SUBAPPLICATION Uebung_003e_AX (* DigitalInput_I1-4 auf DigitalOutput_Q1-4 - flach mit Adapter mit Bypass (Druckumlaufventil) *)
  (* Standard: 61499-2; Description: Copyright (c) 2023 Meisterschulen am Ostbahnhof This program and the accompanying materials are made available under the terms of the Eclipse Public License 2.0 which is available at https://www.eclipse.org/legal/epl-2.0/ SPDX-License-Identifier: EPL-2.0 *)
  (* Version 1.0, 2023-10-23, Franz Höpfinger, Meisterschulen am Ostbahnhof, initial API and implementation and/or initial documentation *)
  PACKAGE Uebungen;
  IMPORT logiBUS::io::DI::logiBUS_DI::Input_I1;
  IMPORT logiBUS::io::DI::logiBUS_DI::Input_I2;
  IMPORT logiBUS::io::DI::logiBUS_DI::Input_I3;
  IMPORT logiBUS::io::DI::logiBUS_DI::Input_I4;
  IMPORT logiBUS::io::DQ::logiBUS_DO::Output_Q1;
  IMPORT logiBUS::io::DQ::logiBUS_DO::Output_Q2;
  IMPORT logiBUS::io::DQ::logiBUS_DO::Output_Q3;
  IMPORT logiBUS::io::DQ::logiBUS_DO::Output_Q4;
  IMPORT logiBUS::io::DQ::logiBUS_DO::Output_Q8;
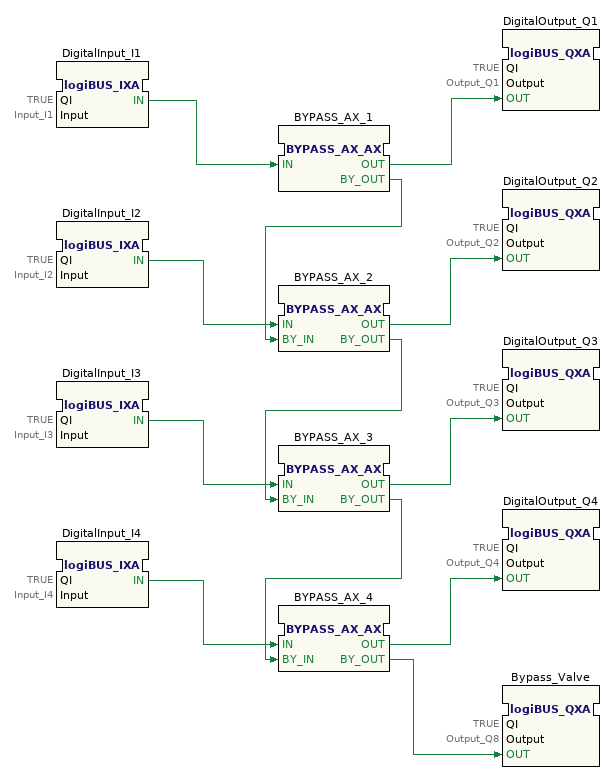
  FBS
    DigitalOutput_Q1 : logiBUS::io::DQ::logiBUS_QXA(QI := TRUE, Output := Output_Q1);
    DigitalInput_I1 : logiBUS::io::DI::logiBUS_IXA(QI := TRUE, Input := Input_I1);
    DigitalOutput_Q2 : logiBUS::io::DQ::logiBUS_QXA(QI := TRUE, Output := Output_Q2);
    DigitalInput_I2 : logiBUS::io::DI::logiBUS_IXA(QI := TRUE, Input := Input_I2);
    BYPASS_AX_1 : logiBUS::signalprocessing::bypass::BYPASS_AX_AX;
    Bypass_Valve : logiBUS::io::DQ::logiBUS_QXA(QI := TRUE, Output := Output_Q8);
    BYPASS_AX_2 : logiBUS::signalprocessing::bypass::BYPASS_AX_AX;
    DigitalOutput_Q3 : logiBUS::io::DQ::logiBUS_QXA(QI := TRUE, Output := Output_Q3);
    DigitalInput_I3 : logiBUS::io::DI::logiBUS_IXA(QI := TRUE, Input := Input_I3);
    BYPASS_AX_3 : logiBUS::signalprocessing::bypass::BYPASS_AX_AX;
    DigitalOutput_Q4 : logiBUS::io::DQ::logiBUS_QXA(QI := TRUE, Output := Output_Q4);
    DigitalInput_I4 : logiBUS::io::DI::logiBUS_IXA(QI := TRUE, Input := Input_I4);
    BYPASS_AX_4 : logiBUS::signalprocessing::bypass::BYPASS_AX_AX;
  END_FBS
  ADAPTER_CONNECTIONS
    DigitalInput_I1.IN TO BYPASS_AX_1.IN;
    BYPASS_AX_1.OUT TO DigitalOutput_Q1.OUT;
    DigitalInput_I2.IN TO BYPASS_AX_2.IN;
    BYPASS_AX_2.OUT TO DigitalOutput_Q2.OUT;
    DigitalInput_I3.IN TO BYPASS_AX_3.IN;
    BYPASS_AX_3.OUT TO DigitalOutput_Q3.OUT;
    DigitalInput_I4.IN TO BYPASS_AX_4.IN;
    BYPASS_AX_4.OUT TO DigitalOutput_Q4.OUT;
    BYPASS_AX_1.BY_OUT TO BYPASS_AX_2.BY_IN;
    BYPASS_AX_2.BY_OUT TO BYPASS_AX_3.BY_IN;
    BYPASS_AX_3.BY_OUT TO BYPASS_AX_4.BY_IN;
    BYPASS_AX_4.BY_OUT TO Bypass_Valve.OUT;
  END_CONNECTIONS
END_SUBAPPLICATION
